Fanuc KAREL source: NC0006.KL

-- PROVISIONAL review KL for V1013-1; original PC SHA256 351639845774201bb6cfb60e710000f1b0ff6fca4ba84229b936f1f1baabb6f5
-- Incomplete behavior may be omitted. Consult companion uncertainty JSON. Do not deploy.
PROGRAM NC0006
%NOLOCKGROUP
-- UNRESOLVED_LOCAL_POOL 1 cells at code offset 3; source declarations unknown
-- DIRECT_LOCAL_WORD_ACCESS alone does not prove INTEGER, REAL, or BOOLEAN
BEGIN
  -- UNRESOLVED_PC offsets 0-8; opcodes 2B,2C,7B
  -- UNRESOLVED_PC offsets 13-20; opcodes 9D,23
  -- UNRESOLVED_PC offsets 25-38; opcodes 21,9D,57,79
  -- UNRESOLVED_PC offsets 43-56; opcodes 21,9D,57,79
  -- UNRESOLVED_PC offsets 61-74; opcodes 21,9D,57,79
  -- UNRESOLVED_PC offsets 79-92; opcodes 21,9D,57,79
  -- UNRESOLVED_PC offsets 97-110; opcodes 21,9D,57,79
  -- UNRESOLVED_PC offsets 115-128; opcodes 21,9D,57,79
  -- UNRESOLVED_PC offsets 133-146; opcodes 21,9D,57,79
  -- UNRESOLVED_PC offsets 151-164; opcodes 21,9D,57,79
  -- UNRESOLVED_PC offsets 169-183; opcodes 21,9D,52,23
  -- UNRESOLVED_PC offsets 188-193; opcodes 7A
  -- UNRESOLVED_PC offsets 198-216; opcodes 21,2E,52,23
  -- UNRESOLVED_PC offsets 226-231; opcodes 7A
  -- UNRESOLVED_PC offsets 236-254; opcodes 21,2E,52,23
  -- UNRESOLVED_PC offsets 264-269; opcodes 7A
  -- UNRESOLVED_PC offsets 274-292; opcodes 21,2E,52,23
  -- UNRESOLVED_PC offsets 302-307; opcodes 7A
  -- UNRESOLVED_PC offsets 312-330; opcodes 21,2E,52,23
  -- UNRESOLVED_PC offsets 340-345; opcodes 7A
  -- UNRESOLVED_PC offsets 350-368; opcodes 21,2E,52,23
  -- UNRESOLVED_PC offsets 378-383; opcodes 7A
  -- UNRESOLVED_PC offsets 388-406; opcodes 21,2E,52,23
  -- UNRESOLVED_PC offsets 416-421; opcodes 7A
  -- UNRESOLVED_PC offsets 426-444; opcodes 21,2E,52,23
  -- UNRESOLVED_PC offsets 454-459; opcodes 7A
  -- UNRESOLVED_PC offsets 464-482; opcodes 21,2E,52,23
  -- UNRESOLVED_PC offsets 492-496; opcodes 7F
  -- UNRESOLVED_PC offsets 501-505; opcodes 27,AA
  -- UNRESOLVED_PC offsets 510-514; opcodes 7F
END NC0006
